// Mitsubishi GX Works2 project: 0715_P_003_buzzer&RestartAdded   PLC: Q03UDV

// global labels: Global1
VAR_GLOBAL
  R흡착기온명령 AT X1000 : BOOL;
  R흡착기오프명령 AT X1001 : BOOL;
  흡착기온솔밸브 AT Y42 : BOOL;
  흡착기오프솔밸브 AT Y43 : BOOL;
  R고정온명령 AT X100A : BOOL;
  R고정오프명령 AT X100B : BOOL;
  고정전솔 AT Y40 : BOOL;
  고정후솔 AT Y41 : BOOL;
  컨베이어_정구동 AT Y48 : BOOL;
  컨베이어_역구동 AT Y49 : BOOL;
  TG1 AT X2A : BOOL;
  TG2 AT X2B : BOOL;
  TG3 AT X2C : BOOL;
  PB4 AT X2D : BOOL;
  PB5 AT X2E : BOOL;
  경광녹색 AT Y44 : BOOL;
  경광황색 AT Y45 : BOOL;
  경광적색 AT Y46 : BOOL;
  부저 AT Y47 : BOOL;
  R컨정구동 AT X1008 : BOOL;
  R컨역구동 AT X1009 : BOOL;
  베이스도착포토 AT X29 : BOOL;
  R베이스도착포토 AT Y100A : BOOL;
  R재공급요청부저 AT X1004 : BOOL;
  R_재시작 AT Y1008 : BOOL;
END_VAR

PROGRAM MAIN
VAR
  컨베이어_정구동신호 : BOOL;
  컨베이어_역구동신호 : BOOL;
  T_재시작리셋타이머 : TIMER;
END_VAR
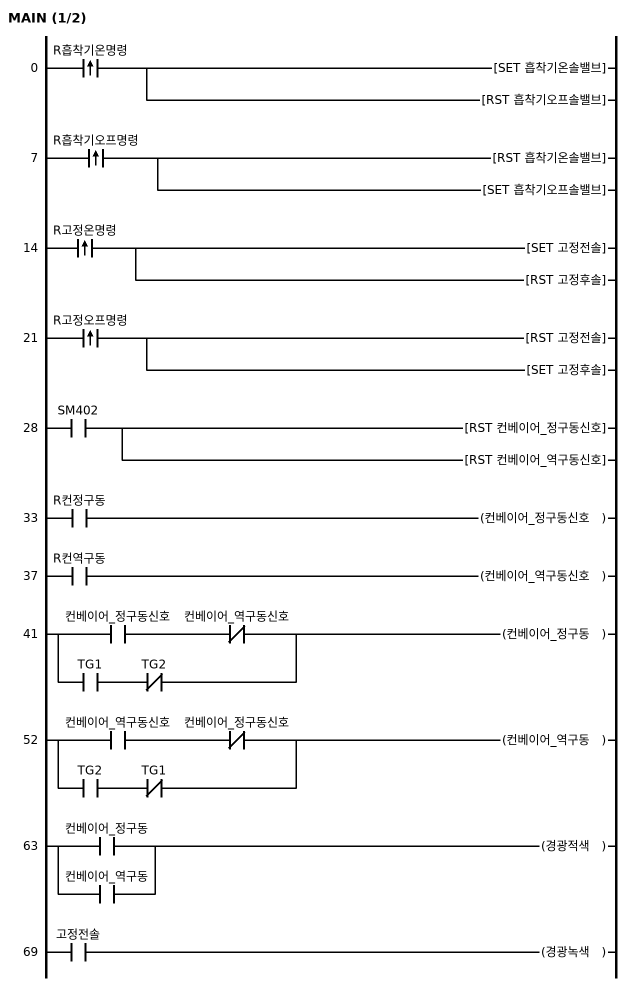
0     LDP     R흡착기온명령
      SET     흡착기온솔밸브
      RST     흡착기오프솔밸브
7     LDP     R흡착기오프명령
      RST     흡착기온솔밸브
      SET     흡착기오프솔밸브
14    LDP     R고정온명령
      SET     고정전솔
      RST     고정후솔
21    LDP     R고정오프명령
      RST     고정전솔
      SET     고정후솔
28    LD      SM402
      RST     컨베이어_정구동신호
      RST     컨베이어_역구동신호
33    LD      R컨정구동
      OUT     컨베이어_정구동신호
37    LD      R컨역구동
      OUT     컨베이어_역구동신호
41    LD      컨베이어_정구동신호
      ANI     컨베이어_역구동신호
      LD      TG1
      ANI     TG2
      ORB
      OUT     컨베이어_정구동
52    LD      컨베이어_역구동신호
      ANI     컨베이어_정구동신호
      LD      TG2
      ANI     TG1
      ORB
      OUT     컨베이어_역구동
63    LD      컨베이어_정구동
      OR      컨베이어_역구동
      OUT     경광적색
69    LD      고정전솔
      OUT     경광녹색
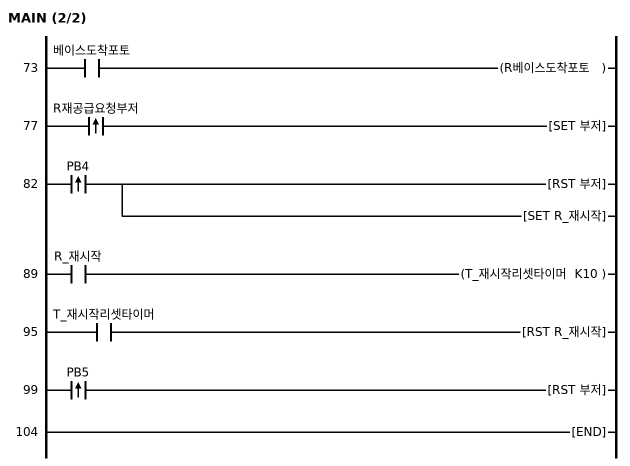
73    LD      베이스도착포토
      OUT     R베이스도착포토
77    LDP     R재공급요청부저
      SET     부저
82    LDP     PB4
      RST     부저
      SET     R_재시작
89    LD      R_재시작
      OUT     T_재시작리셋타이머 K10
95    LD      T_재시작리셋타이머
      RST     R_재시작
99    LDP     PB5
      RST     부저
104   END
END_PROGRAM
